# EPICS substitutions: HUBER/HUBER-IOC-01App/Db/asyn_motor.substitutions
file $(MOTOR)/motorApp/Db/asyn_motor.db {

pattern {P,      N,     M,         DTYP,      PORT,  ADDR,    DESC,        EGU,     DIR,  VELO,  VBAS,  ACCL,  BDST,  BVEL,  BACC,  MRES,  PREC,  DHLM,  DLLM,  INIT}
{"\$(P)", 1, "\$(M)", "asynMotor",  "\$(PORT)",    "\$(ADDR)",  "\$(M) (HUBER)",  mm,  Pos,  1,     0,    .2,    0,     .5,     .2,    0.0001,  6,     0,   0,  ""}
}
